TYPE U_LED :
UNION
	uiUINT		:UINT;
	stLED		:ST_LED;
	
END_UNION
END_TYPE

(* stored: Version 1.1.0.1
   DUT U_LED: Id {141e173f-e1e9-4e4d-917e-f6108e1c60d5} *)
